FUNCTION_BLOCK FB_DIV_DINT (* Divides two DINIT values *)
  (* Standard: 61499-1; Classification: Mathematic; Function: DIVIDER; Type: Mathematical function *)
  (* Version 1.0, 2007-06-26, TS, PROFACTOR GmbH *)
  (* Compiler header: package fb.rt.mathnew; *)
  (* Compiler Java Sun JDK >1.3 *)
  (* Compiler Cpp GNU GCC >3.0 *)
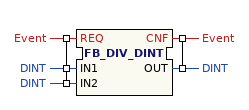
  EVENT_INPUT
    REQ WITH IN1, IN2; (* Normal Execution Request *)
  END_EVENT
  EVENT_OUTPUT
    CNF WITH OUT; (* Execution Confirmation *)
  END_EVENT
  VAR_INPUT
    IN1 : DINT; (* First funtion input *)
    IN2 : DINT; (* Second function input *)
  END_VAR
  VAR_OUTPUT
    OUT : DINT; (* Function output *)
  END_VAR
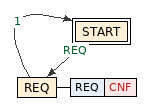
  EC_STATES
    START; (* Initial State *)
    REQ : REQ -> CNF; (* Normal execution *)
  END_STATES
  EC_TRANSITIONS
    START TO REQ := REQ;
    REQ TO START := 1;
  END_TRANSITIONS
  ALGORITHM REQ IN ST: (* Normally executed algorithm *)
OUT:=IN1/IN2;
  END_ALGORITHM
END_FUNCTION_BLOCK
